  rq_init_comm_if_connected(9, "1")
  rq_init_comm_if_connected(2, "2")
  rq_init_comm_if_connected(3, "3")
  rq_init_comm_if_connected(4, "4")
  rq_print_connected_grippers()
  rq_gripper_communication_thread = run rq_gripper_communication()
  set_closed_norm(100.0, 1)
  set_open_norm(0.0, 1)
  set_closed_mm(0.0, 1)
  set_open_mm(50.0, 1)
  set_closed_norm(100.0, 2)
  set_open_norm(0.0, 2)
  set_closed_mm(0.0, 2)
  set_open_mm(50.0, 2)
  set_closed_norm(100.0, 3)
  set_open_norm(0.0, 3)
  set_closed_mm(0.0, 3)
  set_open_mm(50.0, 3)
  set_closed_norm(100.0, 4)
  set_open_norm(0.0, 4)
  set_closed_mm(0.0, 4)
  set_open_mm(50.0, 4)
  rq_current_limit_enabled = False
  while(not rq_gripper_communication_thread_started):
      sleep(0.008)
  end
  # end: URCap Installation Node
  step_count_0a6452fb_7451_455c_a984_e37a8a9f8a68 = 0.0
  thread Step_Counter_Thread_adc0f1ae_8475_4ad6_b4ed_5f883a9c7086():
    while (True):
      step_count_0a6452fb_7451_455c_a984_e37a8a9f8a68 = step_count_0a6452fb_7451_455c_a984_e37a8a9f8a68 + 1.0
      sync()
    end
  end
  run Step_Counter_Thread_adc0f1ae_8475_4ad6_b4ed_5f883a9c7086()
  global Pallet_1_cnt_1=1
  global Pallet_1_cnt_2=1
  global Pallet_1_lct_1=1
  global Pallet_1_lct_2=1
  global Pallet_1_lno_1=1
  global Pallet_1_lno_2=1
  global Pallet_1_sep_1= False
  global Pallet_1_sep_2= False
  global Pallet_1_tct_1=1
  global Pallet_1_tct_2=1
  global Waypoint_1_p=p[.006311202988, -.396731900181, .694709116168, -.017551835463, 2.216342413342, -2.222659985206]
  global Waypoint_1_q=[-0.0061829725848596695, -1.5732938251891078, -0.0015221378998830914, -1.5785185299315394, -1.46214162008107E-4, 0.0057725547812879086]
  global Waypoint_7_p=p[.403615773509, -.021754800857, .128515833288, 2.230189812321, -2.181024304153, .065200721433]
  global Waypoint_7_q=[0.3049320876598358, -1.903140207330221, -1.1731582880020142, -1.6353842220702113, 1.5120816230773926, 0.28998205065727234]
  global Approach_1_p=p[.403610859392, -.021735731100, .128517540769, 2.230228811206, -2.181010787824, .065179304682]
  global Approach_1_q=[0.3049320876598452, -1.9031402073302282, -1.173158288002, -1.6353842220702273, 1.5120816230773793, 0.2899820506572816]
  global ToolActionPoi_1_p=p[.419173511739, -.027417847189, .014219003837, -2.193780400164, 2.182112331449, -.046779182353]
  global ToolActionPoi_1_q=[0.2505807876586914, -2.028933664361471, -1.5665972232818604, -1.0606725972941895, 1.5571714639663696, 0.24598589539527893]
  global Exit_2_p=p[.403617591986, -.021748237917, .128541229143, 2.230255984815, -2.181022346474, .065232647838]
  global Exit_2_q=[0.30493208765984026, -1.9031402073302326, -1.1731582880019928, -1.63538422207023, 1.5120816230773864, 0.28998205065727684]
  global Waypoint_8_p=p[.298989811234, .207505266482, .263539995016, -3.026537464073, -.011179441773, -.037672651985]
  global Waypoint_8_q=[-2.9947667757617396, -1.286858008509018, 0.5869744459735315, -0.9132890862277527, -1.4735482374774378, -1.419941250477926]
  global Waypoint_9_p=p[.408570573302, .160256793504, .184062204585, 3.127048647467, -.003167415511, .102853157027]
  global Waypoint_9_q=[-3.061507527028219, -1.0528925222209473, 0.6730626265155237, -1.2556438010982056, -1.603964630757467, -1.4850652853595179]
  global Waypoint_10_p=p[.298998614455, .207517056080, .263537284521, -3.026508397199, -.011225329479, -.037696689366]
  global Waypoint_10_q=[-2.99475604692568, -1.2868440014174958, 0.5869877974139612, -0.9133362931064148, -1.4735224882708948, -1.419959847127096]
  global Waypoint_11_p=p[.407764802673, .173494233423, .172615162272, -3.118779367809, -.011065957388, -.063563570396]
  global Waypoint_11_q=[-3.053194586430685, -1.031084732418396, 0.6844828764544886, -1.2670062643340607, -1.5672581831561487, -1.485044304524557]
  global Waypoint_12_p=p[.298999820506, .207509261838, .263545985735, -3.026514261686, -.011302718141, -.037745196043]
  global Waypoint_12_q=[-2.994772497807638, -1.2868661147407074, 0.5869792143451136, -0.9133316439441224, -1.4735320250140589, -1.4200261274920862]
  global Waypoint_5_p=p[-.064630700940, -.396800927927, .174762175547, .062127931683, 3.094885185543, .044365086974]
  global Waypoint_5_q=[-1.4395549933062952, -2.008991857568258, -0.7906087636947632, -1.9334246120848597, 1.60926353931427, 0.18173667788505554]
  global Waypoint_6_p=p[-.073197224054, -.437246535759, .079066895105, 2.240473684801, -2.161384789820, -.032207847264]
  global Waypoint_6_q=[-1.4182103315936487, -2.0974489651122035, -1.1174896955490112, -1.4966496539166947, 1.522871494293213, -1.4482644240008753]
  global Waypoint_2_p=p[-.173442394654, -.436915197966, .182927340629, 2.171747879898, -2.164820390506, .003964422445]
  global Waypoint_2_q=[0.9134483337402344, -0.8295380634120484, 0.29382020631899053, -1.1101735097220917, -1.5925639311419886, -2.226902786885397]
  global Waypoint_3_p=p[-.180920881159, -.420236380523, .065873760122, -2.189279979070, 2.222870670837, .015977319260]
  global Waypoint_3_q=[0.8771921992301941, -0.9237610262683411, 0.9896367231952112, -1.6144501171507777, -1.5941713492022913, -2.2494285742389124]
  global Waypoint_4_p=p[-.173450947462, -.436913786129, .182946855856, 2.171686326404, -2.164800772723, .003954388964]
  global Waypoint_4_q=[0.9134395122528076, -0.8295797866633912, 0.29382497469057256, -1.110192672615387, -1.5925777594195765, -2.2268932501422327]
  global Approach_p=p[-.374933253319, -.099241273108, .091187517551, -2.186920108179, -2.181351939136, -.068958068249]
  global Approach_q=[-0.039641682301656544, -1.2695138913444062, 1.4103511015521448, -1.7197658024229945, -1.653177563344137, -0.03747255006899053]
  global ToolActionPoint_p=p[-.388778394884, -.099413998565, .017541197521, -2.201152476360, -2.237622626666, .025746250277]
  global ToolActionPoint_q=[-0.09210378328432256, -1.158921555881836, 1.6148517767535608, -2.0394679508604945, -1.5729945341693323, -0.11253196397890264]
  global Exit_1_p=p[-.374923257911, -.099233247993, .091151097461, -2.187007269407, -2.181421653035, -.069007565653]
  global Exit_1_q=[-0.03970319429506475, -1.2694595617106934, 1.4104049841510218, -1.7197748623290003, -1.6531232039081019, -0.03752261797060186]
  $ 2 "BeforeStart"
  $ 3 "pregunta≔ True "
  global pregunta=  True
  # begin: URCap Program Node
  #   Source: Robotiq_Grippers, 2.4.0.45103, Robotiq Inc.
  #   Type: Gripper
  $ 4 "Gripper Open (1)"
  if not(gripper_connected[0]):
    popup("Gripper 1 must be connected to run this program.", "No connection", False, True, True)
  end
  if not(rq_is_gripper_activated("1")):
    popup("Gripper 1 is not activated. Go to Installation tab > Gripper to activate it and run the program again.", "Not activated", False, True, True)
  end
  rq_set_pos_spd_for(0, 0, 179, "1")
  rq_wait_pos_spe_for_request(0, 0, 179, "1")
  rq_go_to("1")
  rq_wait("1")
  # end: URCap Program Node
  $ 5 "cont≔0"
  global cont=0
  $ 84 "Thread_1"
  thread Thread_1():
    while (True):
      $ 85 "If sensor≟ False "
      if (get_standard_digital_in(0) ==   False  ):
        $ 86 "Set DO[0]=Off"
        set_standard_digital_out(0, False)
      else:
        $ 87 "Else" "noBreak"
        $ 88 "Set DO[0]=On"
        set_standard_digital_out(0, True)
      end
    end
  end
  threadId_Thread_1 = run Thread_1()
  while (True):
    $ 6 "Robot Program"
    $ 7 "MoveJ"
    $ 8 "Waypoint_1" "breakAfter"
    movej(get_inverse_kin(Waypoint_1_p, qnear=Waypoint_1_q), a=1.3962634015954636, v=1.0471975511965976)
    $ 9 "MoveJ"
    $ 10 "Waypoint_7" "breakAfter"
    movej(get_inverse_kin(Waypoint_7_p, qnear=Waypoint_7_q), a=1.3962634015954636, v=1.0471975511965976)
    $ 11 "Pallet_2"
    def Pallet_2_trans(pose):
    return p[pose[0], pose[1], pose[2], 0, 0, 0]
  end
  def Pallet_2_rot(pose):
  return p[0, 0, 0, pose[3], pose[4], pose[5]]
  end
  def Pallet_2_compute_pallet_waypoint(T_base_feature_taught, T_feature_referencePoint_taught, T_referencePoint_approach_taught, T_base_feature, T_base_referencePoint):
  local trans_referencePoint_approach_in_feature_taught = pose_sub(Pallet_2_trans(pose_trans(T_feature_referencePoint_taught, T_referencePoint_approach_taught)), Pallet_2_trans(T_feature_referencePoint_taught))
  local rot_referencePoint_approach_in_feature_taught = pose_trans(Pallet_2_rot(T_feature_referencePoint_taught), pose_trans(Pallet_2_rot(T_referencePoint_approach_taught), pose_inv(Pallet_2_rot(T_feature_referencePoint_taught))))
  T_feature_referencePoint = pose_trans(pose_inv(T_base_feature), T_base_referencePoint)
  rot_referencePoint_approach = pose_trans(pose_inv(Pallet_2_rot(T_feature_referencePoint)), pose_trans(rot_referencePoint_approach_in_feature_taught, Pallet_2_rot(T_feature_referencePoint)))
  T_feature_approach = pose_trans(trans_referencePoint_approach_in_feature_taught, pose_trans(T_feature_referencePoint, rot_referencePoint_approach))
  T_base_approach = pose_trans(T_base_feature, T_feature_approach)
  return T_base_approach
  end
  Pallet_1_tct_1 = 6
  if (Pallet_1_cnt_1 > 6 or Pallet_1_cnt_1 < 1):
    Pallet_1_cnt_1 = 1
  end
  $ 12 "Patterns" "noBreak"
  $ 13 "Grid_Pattern_2" "noBreak"
  $ 18 "Layers" "noBreak"
  if (Pallet_1_cnt_1 < 7):
    Pallet_1_lno_1 = 1
    Pallet_1_lct_1 = Pallet_1_cnt_1
    global CornerItem_5=pose_trans(p[0.0,0.0,0.0,0.0,0.0,0.0], pose_trans(p[-.000000000000, -.000000000000, -.000000000000, .000000000000, .000000000000, .000000000000], p[.419182990657, -.027403329201, .014215626278, -2.193846802957, 2.182049919946, -.046816911117]))
    global CornerItem_6=pose_trans(p[0.0,0.0,0.0,0.0,0.0,0.0], pose_trans(p[-.000000000000, -.000000000000, -.000000000000, .000000000000, .000000000000, .000000000000], p[.316991768671, -.025773753017, .016519811029, 2.253003057016, -2.154543682309, -.011490606798]))
    global CornerItem_7=pose_trans(p[0.0,0.0,0.0,0.0,0.0,0.0], pose_trans(p[-.000000000000, -.000000000000, -.000000000000, .000000000000, .000000000000, .000000000000], p[.320612166659, -.229806400228, .017657793389, -2.244638845679, 2.197166083922, .029638314282]))
    global CornerItem_8=pose_trans(p[0.0,0.0,0.0,0.0,0.0,0.0], pose_trans(p[-.000000000000, -.000000000000, -.000000000000, .000000000000, .000000000000, .000000000000], p[.415810577080, -.229001861117, .016481325028, -2.244187789181, 2.164998044969, -.073546384811]))
    Pallet_1_cnt_1_x = (Pallet_1_lct_1 - 1) % 2
    Pallet_1_cnt_1_y = floor((Pallet_1_lct_1 - 1) / 2)
    referencePoin_1 = interpolate_pose(interpolate_pose(CornerItem_5, CornerItem_6, Pallet_1_cnt_1_x/1), interpolate_pose(CornerItem_8, CornerItem_7,Pallet_1_cnt_1_x/1), Pallet_1_cnt_1_y/2)
    direction = p[0,0,1,0,0,0]
    referencePoin_1 = pose_add (referencePoin_1,p[0.0*direction[0],0.0*direction[1],0.0*direction[2],0,0,0])
  end
  Approach_1_p = Pallet_2_compute_pallet_waypoint(p[0.0,0.0,0.0,0.0,0.0,0.0], pose_trans(pose_inv(p[0.0,0.0,0.0,0.0,0.0,0.0]), p[0.4213113469638263,-0.01819052519312586,0.010406333504865667,2.240112144944265,-2.1778209481181734,0.11345289794319778]), p[0.010459468591118015,0.013104402996390319,-0.11830049520425878,-0.02611798904828491,-0.017639671230119527,0.005416859308159515], p[0.0,0.0,0.0,0.0,0.0,0.0], referencePoin_1)
  Approach_1_p = pose_trans(p[0.4213113469638263,-0.01819052519312586,0.010406333504865667,2.240112144944281,-2.1778209481181885,0.11345289794318614], pose_trans(pose_inv(referencePoin_1), Approach_1_p))
  ToolActionPoi_1_p = Pallet_2_compute_pallet_waypoint(p[0.0,0.0,0.0,0.0,0.0,0.0], pose_trans(pose_inv(p[0.0,0.0,0.0,0.0,0.0,0.0]), p[0.4213113469638263,-0.01819052519312586,0.010406333504865667,2.240112144944265,-2.1778209481181734,0.11345289794319778]), p[0.009387185059632146,0.0022556052084201084,-0.0033231412132662327,0.014395013283138374,-0.07330493640865068,0.024782130658139983], p[0.0,0.0,0.0,0.0,0.0,0.0], referencePoin_1)
  ToolActionPoi_1_p = pose_trans(p[0.4213113469638263,-0.01819052519312586,0.010406333504865667,2.240112144944281,-2.1778209481181885,0.11345289794318614], pose_trans(pose_inv(referencePoin_1), ToolActionPoi_1_p))
  Exit_2_p = Pallet_2_compute_pallet_waypoint(p[0.0,0.0,0.0,0.0,0.0,0.0], pose_trans(pose_inv(p[0.0,0.0,0.0,0.0,0.0,0.0]), p[0.4213113469638263,-0.01819052519312586,0.010406333504865667,2.240112144944265,-2.1778209481181734,0.11345289794319778]), p[0.010473611254511392,0.013097108090575293,-0.11832307078278237,-0.026073702540664042,-0.01763549929069169,0.00541127787852485], p[0.0,0.0,0.0,0.0,0.0,0.0], referencePoin_1)
  Exit_2_p = pose_trans(p[0.4213113469638263,-0.01819052519312586,0.010406333504865667,2.240112144944281,-2.1778209481181885,0.11345289794318614], pose_trans(pose_inv(referencePoin_1), Exit_2_p))
  $ 19 "At Each Item" "noBreak"
  $ 20 "Generated Movements" "noBreak"
  $ 21 "MoveJ" "noBreak"
  $ 22 "Approach_1" "noBreak"
  movej(get_inverse_kin(pose_trans(referencePoin_1, pose_trans(p[-.030131796481, .420675404285, -.008168055752, -2.240112144944, 2.177820948118, -.113452897943], Approach_1_p)), qnear=Approach_1_q), a=1.3962634015954636, v=1.0471975511965976)
  $ 23 "MoveL" "noBreak"
  $ 24 "ToolActionPoi_1" "noBreak"
  movel(pose_trans(referencePoin_1, pose_trans(p[-.030131796481, .420675404285, -.008168055752, -2.240112144944, 2.177820948118, -.113452897943], ToolActionPoi_1_p)), a=1.2, v=0.25)
  $ 25 "Tool action" "noBreak"
  # begin: URCap Program Node
  #   Source: Robotiq_Grippers, 2.4.0.45103, Robotiq Inc.
  #   Type: Gripper
  $ 26 "Gripper Move89% (1)" "noBreak"
  if not(gripper_connected[0]):
    popup("Gripper 1 must be connected to run this program.", "No connection", False, True, True)
  end
  if not(rq_is_gripper_activated("1")):
    popup("Gripper 1 is not activated. Go to Installation tab > Gripper to activate it and run the program again.", "Not activated", False, True, True)
  end
  rq_set_pos_spd_for(226, 0, 245, "1")
  rq_wait_pos_spe_for_request(226, 0, 245, "1")
  rq_go_to("1")
  rq_wait("1")
  # end: URCap Program Node
  $ 27 "MoveL" "noBreak"
  $ 28 "Exit_2" "noBreak"
  movel(pose_trans(referencePoin_1, pose_trans(p[-.030131796481, .420675404285, -.008168055752, -2.240112144944, 2.177820948118, -.113452897943], Exit_2_p)), a=1.2, v=0.25)
  Pallet_1_sep_1 = False
  if (Pallet_1_cnt_1 >= 6):
    Pallet_1_cnt_1 = 1
  else:
    Pallet_1_cnt_1 = Pallet_1_cnt_1 + 1
  end
  $ 29 "cont≔cont+1"
  global cont=cont+1
  $ 30 "If cont≟2"
  if (cont == 2):
    $ 31 "MoveJ"
    $ 32 "Waypoint_8" "breakAfter"
    movej(get_inverse_kin(Waypoint_8_p, qnear=Waypoint_8_q), a=1.3962634015954636, v=1.0471975511965976)
    $ 33 "MoveJ"
    $ 34 "Waypoint_9" "breakAfter"
    movej(get_inverse_kin(Waypoint_9_p, qnear=Waypoint_9_q), a=1.3962634015954636, v=1.0471975511965976)
    # begin: URCap Program Node
    #   Source: Robotiq_Grippers, 2.4.0.45103, Robotiq Inc.
    #   Type: Gripper
    $ 35 "Gripper Open (1)"
    if not(gripper_connected[0]):
      popup("Gripper 1 must be connected to run this program.", "No connection", False, True, True)
    end
    if not(rq_is_gripper_activated("1")):
      popup("Gripper 1 is not activated. Go to Installation tab > Gripper to activate it and run the program again.", "Not activated", False, True, True)
    end
    rq_set_pos_spd_for(0, 0, 217, "1")
    rq_wait_pos_spe_for_request(0, 0, 217, "1")
    rq_go_to("1")
    rq_wait("1")
    # end: URCap Program Node
    $ 36 "MoveJ"
    $ 37 "Waypoint_10" "breakAfter"
    movej(get_inverse_kin(Waypoint_10_p, qnear=Waypoint_10_q), a=1.3962634015954636, v=1.0471975511965976)
    $ 38 "pregunta≔'buena?'"
    global pregunta=request_boolean_from_primary_client("buena?")
    $ 39 "cont≔0"
    global cont=0
    $ 40 "If pregunta≟ False "
    if (pregunta ==   False  ):
      $ 41 "Wait: 1.0"
      sleep(1.0)
    else:
      $ 42 "Else" "noBreak"
      $ 43 "MoveJ"
      $ 44 "Waypoint_11" "breakAfter"
      movej(get_inverse_kin(Waypoint_11_p, qnear=Waypoint_11_q), a=1.3962634015954636, v=1.0471975511965976)
      # begin: URCap Program Node
      #   Source: Robotiq_Grippers, 2.4.0.45103, Robotiq Inc.
      #   Type: Gripper
      $ 45 "Gripper Close (1)"
      if not(gripper_connected[0]):
        popup("Gripper 1 must be connected to run this program.", "No connection", False, True, True)
      end
      if not(rq_is_gripper_activated("1")):
        popup("Gripper 1 is not activated. Go to Installation tab > Gripper to activate it and run the program again.", "Not activated", False, True, True)
      end
      rq_set_pos_spd_for(255, 0, 217, "1")
      rq_wait_pos_spe_for_request(255, 0, 217, "1")
      rq_go_to("1")
      rq_wait("1")
      # end: URCap Program Node
      $ 46 "MoveJ"
      $ 47 "Waypoint_12" "breakAfter"
      movej(get_inverse_kin(Waypoint_12_p, qnear=Waypoint_12_q), a=1.3962634015954636, v=1.0471975511965976)
    end
  else:
    $ 48 "Else" "noBreak"
    $ 49 "Wait: 1.0"
    sleep(1.0)
  end
  $ 50 "If pregunta≟ True "
  if (pregunta ==   True  ):
    $ 51 "MoveJ"
    $ 52 "Waypoint_5" "breakAfter"
    movej(get_inverse_kin(Waypoint_5_p, qnear=Waypoint_5_q), a=1.3962634015954636, v=1.0471975511965976)
    $ 53 "MoveJ"
    $ 54 "Waypoint_6" "breakAfter"
    movej(get_inverse_kin(Waypoint_6_p, qnear=Waypoint_6_q), a=1.3962634015954636, v=1.0471975511965976)
    # begin: URCap Program Node
    #   Source: Robotiq_Grippers, 2.4.0.45103, Robotiq Inc.
    #   Type: Gripper
    $ 55 "Gripper Open (1)"
    if not(gripper_connected[0]):
      popup("Gripper 1 must be connected to run this program.", "No connection", False, True, True)
    end
    if not(rq_is_gripper_activated("1")):
      popup("Gripper 1 is not activated. Go to Installation tab > Gripper to activate it and run the program again.", "Not activated", False, True, True)
    end
    rq_set_pos_spd_for(0, 0, 217, "1")
    rq_wait_pos_spe_for_request(0, 0, 217, "1")
    rq_go_to("1")
    rq_wait("1")
    # end: URCap Program Node
  else:
    $ 56 "Else" "noBreak"
    $ 57 "pregunta≔ True "
    global pregunta=  True
  end
  $ 58 "If sensor≟ False "
  if (get_standard_digital_in(0) ==   False  ):
    $ 59 "MoveJ"
    $ 60 "Waypoint_2" "breakAfter"
    movej(get_inverse_kin(Waypoint_2_p, qnear=Waypoint_2_q), a=1.3962634015954636, v=1.0471975511965976)
    $ 61 "MoveJ"
    $ 62 "Waypoint_3" "breakAfter"
    movej(get_inverse_kin(Waypoint_3_p, qnear=Waypoint_3_q), a=1.3962634015954636, v=1.0471975511965976)
    # begin: URCap Program Node
    #   Source: Robotiq_Grippers, 2.4.0.45103, Robotiq Inc.
    #   Type: Gripper
    $ 63 "Gripper Close (1)"
    if not(gripper_connected[0]):
      popup("Gripper 1 must be connected to run this program.", "No connection", False, True, True)
    end
    if not(rq_is_gripper_activated("1")):
      popup("Gripper 1 is not activated. Go to Installation tab > Gripper to activate it and run the program again.", "Not activated", False, True, True)
    end
    rq_set_pos_spd_for(255, 0, 217, "1")
    rq_wait_pos_spe_for_request(255, 0, 217, "1")
    rq_go_to("1")
    rq_wait("1")
    # end: URCap Program Node
    $ 64 "MoveJ"
    $ 65 "Waypoint_4" "breakAfter"
    movej(get_inverse_kin(Waypoint_4_p, qnear=Waypoint_4_q), a=1.3962634015954636, v=1.0471975511965976)
    $ 66 "Pallet_3"
    def Pallet_3_trans(pose):
    return p[pose[0], pose[1], pose[2], 0, 0, 0]
  end
  def Pallet_3_rot(pose):
  return p[0, 0, 0, pose[3], pose[4], pose[5]]
  end
  def Pallet_3_compute_pallet_waypoint(T_base_feature_taught, T_feature_referencePoint_taught, T_referencePoint_approach_taught, T_base_feature, T_base_referencePoint):
  local trans_referencePoint_approach_in_feature_taught = pose_sub(Pallet_3_trans(pose_trans(T_feature_referencePoint_taught, T_referencePoint_approach_taught)), Pallet_3_trans(T_feature_referencePoint_taught))
  local rot_referencePoint_approach_in_feature_taught = pose_trans(Pallet_3_rot(T_feature_referencePoint_taught), pose_trans(Pallet_3_rot(T_referencePoint_approach_taught), pose_inv(Pallet_3_rot(T_feature_referencePoint_taught))))
  T_feature_referencePoint = pose_trans(pose_inv(T_base_feature), T_base_referencePoint)
  rot_referencePoint_approach = pose_trans(pose_inv(Pallet_3_rot(T_feature_referencePoint)), pose_trans(rot_referencePoint_approach_in_feature_taught, Pallet_3_rot(T_feature_referencePoint)))
  T_feature_approach = pose_trans(trans_referencePoint_approach_in_feature_taught, pose_trans(T_feature_referencePoint, rot_referencePoint_approach))
  T_base_approach = pose_trans(T_base_feature, T_feature_approach)
  return T_base_approach
  end
  Pallet_1_tct_2 = 6
  if (Pallet_1_cnt_2 > 6 or Pallet_1_cnt_2 < 1):
    Pallet_1_cnt_2 = 1
  end
  $ 67 "Patterns" "noBreak"
  $ 68 "Grid_Pattern_3" "noBreak"
  $ 73 "Layers" "noBreak"
  if (Pallet_1_cnt_2 < 7):
    Pallet_1_lno_2 = 1
    Pallet_1_lct_2 = Pallet_1_cnt_2
    global CornerItem_9=pose_trans(p[0.0,0.0,0.0,0.0,0.0,0.0], pose_trans(p[-.000000000000, -.000000000000, -.000000000000, .000000000000, .000000000000, .000000000000], p[-.388781703147, -.099430734940, .017543734124, -2.201062958396, -2.237681591188, .025786611760]))
    global CornerItem_10=pose_trans(p[0.0,0.0,0.0,0.0,0.0,0.0], pose_trans(p[-.000000000000, -.000000000000, -.000000000000, .000000000000, .000000000000, .000000000000], p[-.485340209797, -.103251170278, .017553535595, -2.199207834859, -2.231567232551, .062985305011]))
    global CornerItem_11=pose_trans(p[0.0,0.0,0.0,0.0,0.0,0.0], pose_trans(p[-.000000000000, -.000000000000, -.000000000000, .000000000000, .000000000000, .000000000000], p[-.472976099055, -.294925029075, .015720872819, -2.185984718110, -2.186660452689, .174193528135]))
    global CornerItem_12=pose_trans(p[0.0,0.0,0.0,0.0,0.0,0.0], pose_trans(p[-.000000000000, -.000000000000, -.000000000000, .000000000000, .000000000000, .000000000000], p[-.366541785701, -.297361144406, .016755711899, -2.129790332387, -2.179314548755, -.071102642574]))
    Pallet_1_cnt_2_x = (Pallet_1_lct_2 - 1) % 2
    Pallet_1_cnt_2_y = floor((Pallet_1_lct_2 - 1) / 2)
    referencePoint = interpolate_pose(interpolate_pose(CornerItem_9, CornerItem_10, Pallet_1_cnt_2_x/1), interpolate_pose(CornerItem_12, CornerItem_11,Pallet_1_cnt_2_x/1), Pallet_1_cnt_2_y/2)
    direction = p[0,0,1,0,0,0]
    referencePoint = pose_add (referencePoint,p[0.0*direction[0],0.0*direction[1],0.0*direction[2],0,0,0])
  end
  Approach_p = Pallet_3_compute_pallet_waypoint(p[0.0,0.0,0.0,0.0,0.0,0.0], pose_trans(pose_inv(p[0.0,0.0,0.0,0.0,0.0,0.0]), p[-0.4130588302492224,-0.10484315333726675,0.022310033276196073,-2.227946660116148,-2.1522143069255946,-0.07299261882449298]), p[0.011290404046603461,0.03803131525512071,-0.06822898471170893,0.009179516638724534,0.004478042723611208,-0.031727684758073214], p[0.0,0.0,0.0,0.0,0.0,0.0], referencePoint)
  Approach_p = pose_trans(p[-0.4130588302492224,-0.10484315333726675,0.022310033276196073,-2.2279466601161553,-2.1522143069256017,-0.07299261882449248], pose_trans(pose_inv(referencePoint), Approach_p))
  ToolActionPoint_p = Pallet_3_compute_pallet_waypoint(p[0.0,0.0,0.0,0.0,0.0,0.0], pose_trans(pose_inv(p[0.0,0.0,0.0,0.0,0.0,0.0]), p[-0.4130588302492224,-0.10484315333726675,0.022310033276196073,-2.227946660116148,-2.1522143069255946,-0.07299261882449298]), p[0.005947206395213636,0.02406935574955582,0.005201337081047624,0.01674040211951276,-0.07364983641569947,-0.05057626028908506], p[0.0,0.0,0.0,0.0,0.0,0.0], referencePoint)
  ToolActionPoint_p = pose_trans(p[-0.4130588302492224,-0.10484315333726675,0.022310033276196073,-2.2279466601161553,-2.1522143069256017,-0.07299261882449248], pose_trans(pose_inv(referencePoint), ToolActionPoint_p))
  Exit_1_p = Pallet_3_compute_pallet_waypoint(p[0.0,0.0,0.0,0.0,0.0,0.0], pose_trans(pose_inv(p[0.0,0.0,0.0,0.0,0.0,0.0]), p[-0.4130588302492224,-0.10484315333726675,0.022310033276196073,-2.227946660116148,-2.1522143069255946,-0.07299261882449298]), p[0.011296430995983778,0.03804096193102702,-0.06819208821982586,0.009077599193761039,0.0044221022355256595,-0.0317231229899013], p[0.0,0.0,0.0,0.0,0.0,0.0], referencePoint)
  Exit_1_p = pose_trans(p[-0.4130588302492224,-0.10484315333726675,0.022310033276196073,-2.2279466601161553,-2.1522143069256017,-0.07299261882449248], pose_trans(pose_inv(referencePoint), Exit_1_p))
  $ 74 "At Each Item" "noBreak"
  $ 75 "Generated Movements" "noBreak"
  $ 76 "MoveJ" "noBreak"
  $ 77 "Approach" "noBreak"
  movej(get_inverse_kin(pose_trans(referencePoint, pose_trans(p[.117372349870, .409140449125, .030581792122, 2.227946660116, 2.152214306926, .072992618824], Approach_p)), qnear=Approach_q), a=1.3962634015954636, v=1.0471975511965976)
  $ 78 "MoveL" "noBreak"
  $ 79 "ToolActionPoint" "noBreak"
  movel(pose_trans(referencePoint, pose_trans(p[.117372349870, .409140449125, .030581792122, 2.227946660116, 2.152214306926, .072992618824], ToolActionPoint_p)), a=1.2, v=0.25)
  $ 80 "Tool action" "noBreak"
  # begin: URCap Program Node
  #   Source: Robotiq_Grippers, 2.4.0.45103, Robotiq Inc.
  #   Type: Gripper
  $ 81 "Gripper Open (1)" "noBreak"
  if not(gripper_connected[0]):
    popup("Gripper 1 must be connected to run this program.", "No connection", False, True, True)
  end
  if not(rq_is_gripper_activated("1")):
    popup("Gripper 1 is not activated. Go to Installation tab > Gripper to activate it and run the program again.", "Not activated", False, True, True)
  end
  rq_set_pos_spd_for(0, 0, 0, "1")
  rq_wait_pos_spe_for_request(0, 0, 0, "1")
  rq_go_to("1")
  rq_wait("1")
  # end: URCap Program Node
  $ 82 "MoveL" "noBreak"
  $ 83 "Exit_1" "noBreak"
  movel(pose_trans(referencePoint, pose_trans(p[.117372349870, .409140449125, .030581792122, 2.227946660116, 2.152214306926, .072992618824], Exit_1_p)), a=1.2, v=0.25)
  Pallet_1_sep_2 = False
  if (Pallet_1_cnt_2 >= 6):
    Pallet_1_cnt_2 = 1
  else:
    Pallet_1_cnt_2 = Pallet_1_cnt_2 + 1
  end
  end
  end
end
